{attribute 'OPC.UA.DA.StructuredType' := '1'}
TYPE LOGGING_RECORD :
STRUCT
	FirstDateTime : DATE_AND_TIME; 	
	LastDateTime : DATE_AND_TIME; 	
	Message : ERROR_MESSAGE; 	
	MessageCount : ULINT; 	
END_STRUCT
END_TYPE

(* stored: Version 1.1.0.1
   DUT LOGGING_RECORD: Id {9937d639-5e61-4be0-a85f-df6ea9026991} *)
